FUNCTION_BLOCK FB_ReadCoE

VAR_INPUT
	sNetId			: T_AmsNetId;
	nSlaveAddr		: UINT;
	nIndex			: WORD;
	nIndexOffset	: BYTE;
END_VAR

VAR_OUTPUT
	nParameter		: INT;
	bDoneReading	: BOOL;
	bError			: BOOL;
END_VAR

VAR
	bExecute		: BOOL;
	fbCoERead		: FB_EcCoESDoRead;
	eCoEReadState	: (INIT, TRIGGER, READ, DONE);
END_VAR

CASE eCoEReadState OF
	
	INIT:
		bDoneReading := FALSE;
		bExecute := FALSE;
		eCoEReadState := TRIGGER;
	
	TRIGGER:
		bExecute := TRUE;
		eCoEReadState := READ;
		
	READ:
		fbCoERead(
			sNetId:=sNetId, 
			nSlaveAddr:=nSlaveAddr, 
			nSubIndex:=nIndexOffset, 
			nIndex:=nIndex, 
			pDstBuf:=ADR(nParameter), 
			cbBufLen:=SIZEOF(nParameter), 
			bExecute:=bExecute);
			
		bExecute := NOT bExecute;
		
		IF NOT fbCoeRead.bBusy THEN
			eCoEReadState := DONE;
		END_IF
		
	DONE:
		IF fbCoeRead.bError THEN
			bError := TRUE;
		ELSE
			bError := FALSE;
		END_IF
		bDoneReading := TRUE;
		eCoEReadState := INIT;

END_CASE

END_FUNCTION_BLOCK

(* stored: Version 1.1.0.1, ProductVersion 3.1.4024.9
   POU FB_ReadCoE: Id {069f420b-93e5-431e-93c0-caa251f12ccf}, SpecialFunc None *)
